# EPICS substitutions: viocs/tb_bpms/tb_bpmsApp/Db/bpm.substitutions
file "db/bpm.db" {
    pattern { sector, pos }

        { "02", "" }
        { "03", "-A" }
        { "03", "-B" }
        { "04", "" }
        { "05", "" }
}
